REGION Network 10: Example — Equations
   // ▀▀▀▀▀▀▀▀▀▀▀▀▀▀▀▀▀▀▀▀▀▀▀▀▀▀▀▀▀▀▀▀▀▀▀▀▀▀▀▀▀▀▀▀
   // 
   // TITLE:    EQUATIONS (EXAMPLES)
   // 
   // ▄▄▄▄▄▄▄▄▄▄▄▄▄▄▄▄▄▄▄▄▄▄▄▄▄▄▄▄▄▄▄▄▄▄▄▄▄▄▄▄▄▄▄▄
   // 
   // 
   // 
   // ┌─────────────────────────────────────┐
   // │                                                                                                              100                         │
   // │ SigPercent = (Signal ─ PV_RANGE_MIN) ╳ ---------------------------------------------------------------    │
   // │                    (PV_RANGE_MAX ─ PV_RANGE_MIN)    │
   // └─────────────────────────────────────┘
   // 
   // 
   // ┌───────────────────────┐
   // │        2.5               │
   // │ CalcValOOR = ------------ ╳ (RAW_MAX ─ RAW_MIN)   │
   // │       100               │
   // └───────────────────────┘
   // 
   // Mathematical operators:
   //    Large:  ┼ ─ ╳
   //    Small: + − × ÷ ± ≤ ≥
   // 
   //                ━━━   ⬙⬙⬙⬙⬙⬙   ━━━
   // 
   // 
   // ██████████████ █ █ █ █  END   █ █ █ █ ██████████████
END_REGION

REGION Network 11: Example — Figures
   // ▀▀▀▀▀▀▀▀▀▀▀▀▀▀▀▀▀▀▀▀▀▀▀▀▀▀▀▀▀▀▀▀▀▀▀▀▀▀▀▀▀▀▀▀
   // 
   // TITLE:    FIGURES (EXAMPLES)
   // 
   // ▄▄▄▄▄▄▄▄▄▄▄▄▄▄▄▄▄▄▄▄▄▄▄▄▄▄▄▄▄▄▄▄▄▄▄▄▄▄▄▄▄▄▄▄
   // 
   // 
   // 
   // Some example figures, always pad gaps with an EM-SPACE, where text is used add normal 
   // spaces with either a THREE-PER-EM space or a SIX-PER-EM space — one of these will give an
   // exact alignment.
   // 
   // These figures are included to show what is possible.
   // 
   // 
   // Figures have 1 blank line above and 1 below.
   // 
   //   → ┌────────┐
   // ┌───┤   IDLE   │
   // │   └───┬────┘
   // │       ↓
   // │       START
   // │       │
   // │   ┌───┴────┐ →
   // │   │  STARTING     ├───┐
   // │   └───┬────┘   │
   // │       ↓        │
   // │         Run*       ├────────────────────┐
   // │       │        │                    │
   // │   ┌───┴────┐ → │                    │
   // │   │        ├───┴───  Hold  ───┐          │
   // │   │        │             ↓          ↓
   // │   │        │         ┌───┴────┐ ┌───┴────┐
   // │   │        │         │  HOLDING    │ │ ErrHOLDING   │
   // │   │        │         └───┬────┘ └───┬────┘
   // │   │        │             Held*        ErrHeld*
   // │   │        │         ┌───┴────┐ ┌───┴────┐
   // │   │        │         │   HELD    │ │  ErrHELD   │
   // │   │  RUNNING     │         └───┬────┘ └───┬────┘
   // │   │        │              Resume         ErrResume
   // │   │        │         ┌───┴────┐ ┌───┴────┐
   // │  ┌┤        │         │   RESUMING    │ │  ErrRESUMING   │ 
   // │  ││        │         └───┬────┘ └───┬────┘  
   // │  ││        │             │          │
   // │  ││        │ ←           ↓          ↓
   // │  ││        │─────────────┴──────────┘
   // │  │└───┬────┘   Returns to previous step (running or starting)
   // │  ↓    ↓
   // │  │    │
   // │ Complete Complete*     Note: *indicates that the command is issued
   // │  │    │           automatically by the sequence (it
   // │  │┌───┴────┐      can also be triggered manually):
   // │  └┤ COMPLETING  │          1. Run
   // │   └───┬────┘          2. Complete
   // │       ↓               3. Completed
   // ↑     Completed*              4. Held
   // │       │               5. ErrHeld
   // │   ┌───┴────┐          6. Stopped
   // │   │  COMPLETED   │          7. Aborted
   // │   └───┬────┘
   // │       │
   // │              RetIdle*
   // │   ←   ↓
   // ├───────┘
   // │   
   // │
   // │     ABORT ROUTE                  STOPPING ROUTE
   // │Can be triggered in all states except       Can be triggered in all states except
   // │ IDLE, COMPLETED, ABORTING or            IDLE, COMPLETED, ABORTING, 
   // │       ABORTED                 ABORTED, STOPPING or STOPPED
   // │       │                       │
   // │       ↓                       ↓
   // │                Abort                                                                                       Stop
   // │       │                       │
   // │   ┌───┴────┐              ┌───┴────┐
   // ↑   │ ABORTING    │              │  STOPPING    │
   // │   └───┬────┘              └───┬────┘
   // │       ↓                       ↓
   // │              Aborted*                                                                                Stopped*
   // │       │                       │
   // │   ┌───┴────┐              ┌───┴────┐
   // │   │ ABORTED      │              │ STOPPED   │
   // │   └───┬────┘              └───┬────┘
   // │       │                       │
   // │      RetIdle (*)                                                                               RetIdle (*)
   // │  ←    ↓                       ↓
   // └───────┴───────────────────────┘
   // 
   // 
   // 
   // ▌▌▌▌▌▌▌▌▌▌▌▌▌▌▌▌▌▌   INLINE FIGURES ▐▐▐▐▐▐▐▐▐▐▐▐▐▐▐▐▐▐
   // 
   // 
   // 
   // ▂▂▂▂▂▂▂▂▂▂▂▂▂▂▂▂▂▂▂▂▂▂▂▂▂▂▂▂▂▂▂▂▂▂▂▂▂▂▂▂▂▂▂▂
   // 1.1     Step operation and phases
   // 
   // 
   //  ┌─────┐  The sequence progresses from one step to the next if the
   //  │Step n        │  transition logic for the step is TRUE. 
   //  └┬────┘                                                                 
   //   │       In this example, STEP n is active and will remain active
   //         --- T n        until its associated transition (T n) becomes TRUE; at this
   //   │       point the sequence will advance to the next step (STEP n+1)
   //  ┌┴────┐  and execute the actions required of this step. The sequence
   //  │Step n+1    │  will remain in this step until its transition condition is
   //  └┬────┘  true, at which point the sequence will advance again.
   //   │                                                                      
   //         --- T n+1      Each step has a step number, this is an integer value in
   //   │       the range 0 to 29999; step numbers are assigned in specific
   //           Ranges for different operating states of the sequence (IDLE,
   //           STARTING, RUNNING &c.).
   // 
   // Within an individual step, the step has three distinct phases and actions can 
   // be attached to any of these phases (externally to the block). The phases are:
   // 
   // INITIALISING (Phs_INIT)                   ┌──────┐
   // This is activated for a single OB1 scan when the step   │INITIALISING   │
   // is first processed (I.e. on the rising edge of the step     └┬─────┘
   // becoming active).                     │      
   //                           ┌┴─────┐ 
   // PROCESSING (Phs_PROC)               │PROCESSING │
   // This is the main phase of the step, it is activated        └┬─────┘
   // immediately following the INITIALISING phase and remains  │       
   // active until the step TRANSITION condition is TRUE. The     --- T n   
   // PROCESSING phase becomes inactive on the rising edge   │     
   // of the TRANSITION condition.              ┌┴─────┐
   //                           │TERMINATING │    
   // TERMINATING (Phs_TERM)               └──────┘    
   // The TERMINATING phase is activated on the rising edge of the TRANSITION
   // condition (the same condition that terminates the PROCESSING phase). The
   // terminating phase is active for a single OB1 scan.
   // 
   // 
   // [ALTERNATIVE]
   //  ┌──────┐ INITIALISING (Phs_INIT)
   //  │INITIALISING   │ This is activated for a single OB1 scan when the step
   //  └┬─────┘ is first processed (I.e. on the rising edge of the step
   //   │       becoming active).
   //  ┌┴─────┐    
   //  │PROCESSING │ PROCESSING (Phs_PROC)
   //  └┬─────┘ This is the main phase of the step, it is activated 
   //   │       immediately following the INITIALISING phase and remains
   //          --- T n       active until the step TRANSITION condition is TRUE. The
   //   │       PROCESSING phase becomes inactive on the rising edge
   //  ┌┴─────┐ of the TRANSITION condition.
   //  │TERMINATING │    
   //  └──────┘
   // 
   // TERMINATING (Phs_TERM)
   // The TERMINATING phase is activated on the rising edge of the TRANSITION
   // condition (the same condition that terminates the PROCESSING phase). The
   // terminating phase is active for a single OB1 scan.
   // 
   // 
   // 
   // 
   // ▌▌▌▌▌▌▌▌▌▌▌▌▌▌▌▌▌   GRAPHICAL FIGURE   ▐▐▐▐▐▐▐▐▐▐▐▐▐▐▐▐▐
   // 
   //     No. of scans from start of STEP 1
   //     1      2      3     4      5     6       7      8      9
   //   ┼─┼─┼─┼─┼─┼─┼─┼─┼─┼─┼─┼  ─ ─ ┐
   //                                │
   //   ┌─┐                          │
   //   │ │               Phs_INIT
   //  ─┘ └────────────────────                   
   //   ┼─┼─┼─┼─┼─┼─┼─┼─┼─┼─┼─┼                   
   //  
   //     ┌───┐                       S
   //     │   │           Phs_PROC      T
   //  ───┘   └────────────────       E
   //   ┼─┼─┼─┼─┼─┼─┼─┼─┼─┼─┼─┼       P
   //  
   //         ┌─┐                     1
   //         │ │         TRANSITION
   //  ───────┘ └──────────────
   //   ┼─┼─┼─┼─┼─┼─┼─┼─┼─┼─┼─┼
   // 
   //         ┌─┐
   //         │ │         Phs_TERM      │
   //  ───────┘ └──────────────      │
   //   ┼─┼─┼─┼─┼─┼─┼─┼─┼─┼─┼─┼  ─ ─ ┘
   // 
   // 
   //     1      2      3     4      5     6       7      8      9
   //   ┼─┼─┼─┼─┼─┼─┼─┼─┼─┼─┼─┼  ─ ─ ┐
   //                                │
   //           ┌─┐                  │
   //           │ │       Phs_INIT
   //   ────────┘ └────────────                   
   //   ┼─┼─┼─┼─┼─┼─┼─┼─┼─┼─┼─┼                   
   // 
   //             ┌───┐               S
   //             │   │   Phs_PROC      T
   //  ───────────┘   └────────       E
   //   ┼─┼─┼─┼─┼─┼─┼─┼─┼─┼─┼─┼       P
   //                           
   //                 ┌─┐             2
   //                 │ │ TRANSITION
   //  ───────────────┘ └──────      
   //   ┼─┼─┼─┼─┼─┼─┼─┼─┼─┼─┼─┼
   // 
   //                 ┌─┐
   //                 │ │ Phs_TERM      │
   //  ───────────────┘ └──────      │
   //   ┼─┼─┼─┼─┼─┼─┼─┼─┼─┼─┼─┼  ─ ─ ┘
   // 
   // 
   // 
   // ▌▌▌▌▌▌▌▌▌▌▌▌▌▌▌▌▌▌    PAL LOGO    ▐▐▐▐▐▐▐▐▐▐▐▐▐▐▐▐▐▐
   // 
   //          ⠀⠀⠀⠀⠀⠀⠀⠀⠀⠀⠀⠀⠀⠀⠀⠀⠀⠀⠀⠀⠀⠀⠀⠀⠀⠀⠀⠀⠀⣀⣀⣀
   //       ⠀⠀⠀⠀⠀⠀⠀⠀⠀⠀⠀⠀⠀⠀⠀⠀⠀⠀⠀⠀⠀⠀⠀⠀⠀⠀⠀⣤⣶⣿⣿⣿⣿⣿⣿⣤
   //       ⠀⠀⠀⠀⠀⠀⠀⠀⠀⠀⠀⠀⠀⠀⠀⠀⠀⠀⠀⠀⠀⠀⠀⠀⠀⠀⣶⣿⣿⣿⣿⣿⣿⣿⣿⣿⣶
   //       ⠀⠀⠀⠀⠀⠀⠀⠀⠀⠀⠀⠀⠀⠀⠀⠀⠀⠀⠀⠀⠀⠀⠀⠀⠀⠀⣿⣿⣿⣿⣿⣿⣿⣿⣿⣿⣿
   //       ⠀⠀⠀⠀⠀⠀⠀⠀⠀⠀⠀⠀⠀⠀⠀⠀⠀⠀⠀⠀⠀⠀⠀⠀⠀⣀⠛⣿⣿⣿⣿⣿⣿⣿⣿⣿⠿
   //       ⠀⠀⠀⠀⠀⠀⠀⠀⠀⠀⠀⠀⠀⠀⠀⠀⠀⠀⠀⠀⠀⠀⣀⣶⣿⣿⣤⠉⠿⣿⣿⣿⣿⣿⠿⠛⣤⣶
   //       ⠀⠀⠀⠀⠀⠀⠀⠀⠀⠀⠀⠀⠀⠀⠀⠀⠀⠀⠀⠀⣤⣿⣿⣿⣿⣿⣿⣿⣶⣤⠉⠉⠉⠀⠤⣿⣿⣿⣿⣶⣀⣀⣀⣀⣀⣀⣀⣀
   //       ⠀⠀⠀⠀⠀⠀⠀⠀⠀⠀⠀⠀⠀⠀⠀⠀⠀⣀⣶⣿⣿⣿⣿⣿⣿⣿⣿⣿⣿⠉⠀⠀⠀⠀⠀⠉⠿⣿⣿⣿⣿⣿⣿⣿⣿⣿⣿⣿⣶
   //       ⠀⠀⠀⠀⠀⠀⠀⠀⠀⠀⠀⠀⠀⠀⠀⠀⠛⠿⣿⣿⣿⣿⣿⣿⣿⣿⣿⠿⠀⠀⠀⠀⠀⠀⠀⠀⠀⣿⣿⣿⣿⣿⣿⣿⣿⠿⠿⣿⣿⣤
   //       ⠀⠀⠀⠀⠀⠀⠀⠀⠀⣀⣤⣶⣿⣿⣿⣿⣶⣶⣤⠉⠿⣿⣿⣿⣿⣿⠛⠀⠀⠀⠀⠀⠀⠀⠀⠀⠀⣿⣿⣿⣿⠉⠀⠀⠀⠀⠀⠉⣿⣿⣤
   //       ⠀⠀⠀⠀⠀⠀⠀⣀⣶⣿⣿⣿⣿⣿⣿⣿⣿⣿⣿⣿⣤⠉⣿⣿⣿⠛⠀⠀⠀⠀⠀⠀⠀⠀⠀⠀⣿⣿⣿⣿⣿⠀⠀⠀⠀⠀⠀⠀⠀⠿⠿
   //       ⠀⠀⠀⠀⠀⠀⣀⣿⣿⣿⣿⣿⣿⣿⣿⣿⣿⣿⣿⣿⣿⣿⠀⣿⠉⠀⠀⠀⠀⠀⠀⠀⠀⠀⠀⠀⣿⣿⣿⣿⣿
   //       ⠀⠀⠀⠀⠀⠀⣿⣿⣿⣿⣿⣿⣿⣿⣿⣿⣿⣿⣿⣿⣿⣿⣀⠀⠀⠀⠀⠀⠀⠀⠀⠀⠀⠀⠀⠀⠉⠛⠿⣿⣿⣿⣤
   //       ⠀⠀⠀⠀⠀⠀⣿⣿⣿⣿⣿⣿⣿⣿⣿⣿⣿⣿⣿⣿⣿⣿⠿⠀⠀⠀⠀⠀⠀⠀⠀⠀⠀⠀⠀⠀⠀⠀⠀⠀⠉⠛⠿⣿
   //       ⠀⠀⠀⠀⠀⠀⠛⣿⣿⣿⣿⣿⣿⣿⣿⣿⣿⣿⣿⣿⣿⣿
   //       ⠀⠀⠀⠀⠀⠀⠀⠛⣿⣿⣿⣿⣿⣿⣿⣿⣿⣿⣿⣿⠿⠉
   //       ⠀⠀⠀⠀⠀⠀⠀⠀⠀⠛⠿⣿⣿⣿⣿⣿⣿⣿⠿⠉
   //       ⠀⠀⠀⠀⠀⠀⠀⠀⠀⠀⠀⣀⣉⣉⣉⣉⣉⣀
   //       ⠀⠀⠀⠀⠀⠀⠀⠀⠀⣤⣿⣿⣿⣿⣿⣿⣿⣿⣀⠛⣿⣿⣿⣿⣿⣿⣿⣿⣿⣿⣿⣿⣿⣿⣿⣿⣿⣿⣿⣿⣿⣿⣿⣿⣿⣿⣿⣿⣿⣶⣤⣀⠀⠀⠀⠀
   //       ⠀⠀⠀⠀⠀⠀⠀⠀⣤⣿⣿⣿⠿⠉⠉⣿⣿⣿⣿⣤⠉⠿⠿⠿⠿⠿⠿⠿⠿⠿⠿⠿⠿⠿⠿⠿⠿⠿⠿⠿⠿⠿⠿⠿⠿⠿⠿⣿⣿⣿⣿⣿⣿⣀⠀⠀
   //       ⠀⠀⠀⠀⠀⠀⠀⣶⣿⣿⣿⠛⠀⠀   ⠀⠀⠿⣿⣿⣿⣤⠀⠀⠀⠀⠀⠀⣶⣶⣶⣶⣤⠀⠀⠀⠀ ⣶⣶⣶         ⣶⣶⠀⠀⠀⠀⠀⠿⣿⣿⣿⣿⣶⠀
   //       ⠀⠀⠀⠀⠀⠀⣿⣿⣿⣿⠛⠀⠀⠀⠀   ⠀⠀⠛⣿⣿⣿⣶⠀⠀⠀⠀⠀⣿⣿⣿⠿⣿⣿⠀⠀⣤⣿⣿⣿⣤       ⣿⣿⠀⠀⠀⠀⠀⠀ ⠿⣿⣿⣿⣿⣤
   //       ⠀⠀⠀⠀⠀⣿⣿⣿⣿⠉⠀⠀⠀⠀⠀   ⠀⠀⠀⠛⣿⣿⣿⣿⠀⠀⠀⠀⣿⣿⣿⣶⣿⣿⠀⠀⣿⣿⠉⣿⣿       ⣿⣿⠀⠀⠀⠀⠀     ⣿⣿⣿⣿⣿
   //       ⠀⠀⠀⣀⣿⣿⣿⣿⠉⠀⠀⠀⠀⠀⠀⠀⠀   ⠀⠀⠉⣿⣿⣿⣿      ⣿⣿⣿⠛⠛⠀⠀⣶⣿⣿⣿⣿⣿⣶    ⣿⣿⣤⣤⣤      ⣶⣿⣿⣿⣿⠛
   //       ⠀⠀⣤⣿⣿⣿⣿⠉⠀⠀⠀⠀⠀⠀⠀⠀⠀⠀⠀   ⠀⠉⣿⣿⣿⣿⣀ ⠿⠿⠿⠀⠀⠀   ⠿⠿⠉⠉⠉⠿⠿    ⠿⠿⠿⠿⠿ ⠀⣶⣿⣿⣿⣿⠿⠀
   //       ⠀⣤⣿⣿⣿⣿⣿⣶⣤⣤⣤⣤⣤⣤⣤⣤⣤⣤⣤⣤⣶⣿⣿⣿⣿⣿⣀⠀⣶⣶⣶⣶⣶⣶⣶⣶⣶⣶⣶⣶⣶⣶⣶⣶⣶⣶⣶⣶⣿⣿⣿⣿⠉⠀⠀
   //       ⠀⣿⣿⣿⣿⣿⣿⣿⣿⣿⣿⣿⣿⣿⣿⣿⣿⣿⣿⣿⣿⣿⣿⣿⣿⣿⣿⠀⠉⣿⣿⣿⣿⣿⣿⣿⣿⣿⣿⣿⣿⣿⣿⣿⣿⣿⣿⣿⣿⠿⠛⠉⠀⠀⠀⠀
   //       ⠀⠉⠛⠛⠛⠛⠛⠛⠛⠛⠛⠛⠛⠛⠛⠛⠛⠛⠛⠛⠛⠛⠛⠛⠛⠛⠉⠀⠀⠉⠉⠉⠉⠉⠉⠉⠉⠉⠉⠉⠉⠉⠉⠉⠉⠉⠉⠉⠀⠀⠀⠀⠀⠀⠀⠀
   // 
   //                ━━━   ⬙⬙⬙⬙⬙⬙   ━━━
   // 
   // 
   // ██████████████ █ █ █ █  END   █ █ █ █ ██████████████
END_REGION

REGION Network 12: Special characters — Hyphens, whitespace and construction lines
   // ▀▀▀▀▀▀▀▀▀▀▀▀▀▀▀▀▀▀▀▀▀▀▀▀▀▀▀▀▀▀▀▀▀▀▀▀▀▀▀▀▀▀▀▀
   // 
   // TITLE:    SPECIAL CHARACTERS
   // 
   // ▄▄▄▄▄▄▄▄▄▄▄▄▄▄▄▄▄▄▄▄▄▄▄▄▄▄▄▄▄▄▄▄▄▄▄▄▄▄▄▄▄▄▄▄
   // 
   // 
   // The TIA Portal Basic font contains many different types of characters:
   // 
   //    •   Hyphens and whitespace characters
   //    •   Construction lines (these are specially ordered characters, useful for building tables &c.)
   //    •   Arrows
   //    •   Box characters (for drawing box and line diagrams)
   //    •   Block characters
   //    •   Currency
   //    •   Punctuation (extended list)
   //    •   Non-proportional letters and numbers
   //    •   Greek characters
   //    •   Indexing characters
   //    •   Roman numerals
   //    •   Mathematical characters
   //    •   Geometric characters
   //    •   Dingbat characters
   // 
   // The following sections contain a list of these characters for use in TIA Portal comment fields.
   // 
   // Note:    The following tables of characters break the rules for comment fields by exceeding
   //      the prescribed comment field width of 44 em-spaces. This is done to give the 
   //      characters in a more concise form whilst maintaining reasonable descriptions for
   //      the characters
   // 
   // 
   // 
   // ▄▄▄▄▄▄▄▄▄▄▄▄▄▄▄▄▄▄▄▄▄▄▄▄▄▄▄▄▄▄▄▄▄▄▄▄▄▄▄▄▄▄▄▄
   // HYPHENS AND WHITESPACE CHARACTERS
   // 
   // 
   // — Em Dash               █ █ Em Space
   // –   En Dash              █ █   En Space
   // ‐    Hyphen               █ █    Three-Per-Em Space
   // ¬   Soft Hyphen             █ █    Normal Space
   //                       █ █     Six-Per-Em Space
   // 
   // 
   // 
   // ▄▄▄▄▄▄▄▄▄▄▄▄▄▄▄▄▄▄▄▄▄▄▄▄▄▄▄▄▄▄▄▄▄▄▄▄▄▄▄▄▄▄▄▄
   // CONSTRUCTION LINES AND USEFUL LINES
   // 
   // 
   // [Copyable whitespace]
   //  █ █ █ █ █ Em En ThreePerEm SixPerEM
   // [Em-space construction line]
   // ▀▄▀▄▀▄▀▄▀▄▀▄▀▄▀▄▀▄▀▄▀▄▀▄▀▄▀▄▀▄▀▄▀▄▀▄▀▄▀▄▀▄▀▄
   // [Central header — used for examples]
   // ▌▌▌▌▌▌▌▌▌▌▌▌▌▌▌▌▌▌▌▌▌▌▐▐▐▐▐▐▐▐▐▐▐▐▐▐▐▐▐▐▐▐▐▐
   // [Title start]
   // ▀▀▀▀▀▀▀▀▀▀▀▀▀▀▀▀▀▀▀▀▀▀▀▀▀▀▀▀▀▀▀▀▀▀▀▀▀▀▀▀▀▀▀▀
   // [Title end/section over-line]
   // ▄▄▄▄▄▄▄▄▄▄▄▄▄▄▄▄▄▄▄▄▄▄▄▄▄▄▄▄▄▄▄▄▄▄▄▄▄▄▄▄▄▄▄▄
   // [Subsection over-line]
   // ▂▂▂▂▂▂▂▂▂▂▂▂▂▂▂▂▂▂▂▂▂▂▂▂▂▂▂▂▂▂▂▂▂▂▂▂▂▂▂▂▂▂▂▂
   // [Inline section over-line]
   // ▁▁▁▁▁▁▁▁▁▁▁▁▁▁▁▁▁▁▁▁▁▁▁▁▁▁▁▁▁▁▁▁▁▁▁▁▁▁▁▁▁▁▁▁
   // [Table row line]
   //  ――――――――――――――――――――――――――――――――――――――――――
   // [Revision row line]
   //  ―――――――――――――――――――――――――――――――――――――――――――
   // [Flourish divider]
   //                ━━━   ⬙⬙⬙⬙⬙⬙   ━━━
   // [End line]
   // ██████████████ █ █ █ █  END   █ █ █ █ ██████████████
END_REGION

REGION Network 13: Special characters — Arrows, box and block characters
   // ▄▄▄▄▄▄▄▄▄▄▄▄▄▄▄▄▄▄▄▄▄▄▄▄▄▄▄▄▄▄▄▄▄▄▄▄▄▄▄▄▄▄▄▄
   // ARROWS
   // 
   // 
   // ← Left Arrow              ⇐ Left dbl Arrow             ↩ Left Arrow Hook
   // ↑ Up Arrow               ⇑ Up dbl Arrow               ↪ Right Arrow Hook
   // → Right Arrow              ⇒ Right dbl Arrow           ⤣ North West Arrow Hook
   // ↓ Down Arrow             ⇓ Down dbl Arrow             ⤤ North East Arrow Hook
   // ↔ Left Right Arrow             ⇔ Left Right dbl Arrow          ⤥ South East Arrow Hook
   // ↕ Up Down Arrow          ⇕ Up Down dbl Arrow          ⤦ South West Arrow Hook
   // ↖ North West Arrow          ⇖ North West dbl Arrow         ↰    Up Arrow Tip Left
   // ↗ North East Arrow          ⇗ North East dbl Arrow          ↱    Up Arrow Tip Right
   // ↘ South East Arrow          ⇘ South East dbl Arrow         ↲    Down Arrow Tip Left
   // ↙ South West Arrow         ⇙    South West dbl Arrow        ↳ Down Arrow Tip Right
   // ⤡ North West & South East Arrow    ⤂ Left dbl Arrow vert Stroke       ↴ Right Arrow Corner down
   // ⤢ North East & South West Arrow    ⤃ Right dbl Arrow vert Stroke     ↵ Down Arrow Corner Left
   // ⇄ Right Arrow Over Left Arrow       ⤆ Left dbl Arrow From Bar        ↶ Anticlockwise Top Semicircle Arrow
   // ⇅ Up Arrow Left Of down Arrow        ⤇ Right dbl Arrow From Bar         ↷ Clockwise Top Semicircle Arrow
   // ⇆ Left Arrow Over Right Arrow       ⤄ Left Right dbl Arrow vert Stroke    ↺ Anticlockwise Open Circle Arrow
   // ⇇ Left Paired Arrows           ↼ Left Harpoon Barb up         ↻ Clockwise Open Circle Arrow
   // ⇈ Up Paired Arrows             ↽ Left Harpoon Barb down         ⟲ Anticlockwise Gapped Circle Arrow
   // ⇉ Right Paired Arrows         ↾ Up Harpoon Barb Right         ⟳ Clockwise Gapped Circle Arrow
   // ⇊ Down Paired Arrows           ↿ Up Harpoon Barb Left
   // ↤ Left Arrow From Bar           ⇀ Right Harpoon Barb up         ▲  Black Up Triangle 
   // ↥ Up Arrow From Bar          ⇁ Right Harpoon Barb down       ▼  Black Down Triangle
   // ↦ Right Arrow From Bar         ⇂ Down Harpoon Barb Right      ▶  Black Right Triangle
   // ↧ down Arrow From Bar        ⇃ Down Harpoon Barb Left         ◀  Black Left Triangle
   // ↨ Up Down Arrow Base         ⇋ Left Harpoon Over Right Harpoon
   // ↞ Left Two head Arrow          ⇌ Right Harpoon Over Left Harpoon
   // ↟ up Two head Arrow         ↯ Down Zigzag Arrow
   // ↠ Right Two head Arrow
   // ↡ Down Two head Arrow
   // ⤙ Left Arrow-Tail
   // ⤚ Right Arrow-Tail
   // ⤛ Left dbl Arrow-Tail    
   // ⤜ Right dbl Arrow-Tail    
   // ⤝ Left Arrow To Black Diamond    
   // ⤞ Right Arrow To Black Diamond    
   // 
   // ⟵  Long Left Arrow             ↢ Left Arrow Tail             ⌃   Up Arrowhead
   // ⟶  Long Right Arrow          ↣ Right Arrow Tail             ⌄   Down Arrowhead
   // ⟷  Long Left Right Arrow         ⤟ Left Arrow Bar To Black Diamond   ⌅   Projective
   // ⟸  Long Left dbl Arrow         ⤠ Right Arrow Bar To Black Diamond    ⌆   Perspective
   // ⟹  Long Right dbl Arrow          ⤌    Left dbl Dash Arrow         ⟰ Up Quadruple Arrow
   // ⟺  Long Left Right dbl Arrow        ⤍    Right dbl Dash Arrow         ⟱ Down Quadruple Arrow
   // ⟻  Long Left Arrow From Bar       ⤎    Left Triple Dash Arrow        ⤊ Up Triple Arrow
   // ⟼  Long Right Arrow From Bar        ⤏    Right Triple Dash Arrow         ⤋ Down Triple Arrow
   // ⟽  Long Left dbl Arrow From Bar       ⤈    Down Arrow horiz Stroke          ⤈   Down Arrow horiz Stroke
   // ⟾  Long Right dbl Arrow From Bar    ⤉    Up Arrow horiz Stroke             ⤉   Up Arrow horiz Stroke
   // 
   // 
   // 
   // ▄▄▄▄▄▄▄▄▄▄▄▄▄▄▄▄▄▄▄▄▄▄▄▄▄▄▄▄▄▄▄▄▄▄▄▄▄▄▄▄▄▄▄▄
   // BOX CHARACTERS
   // 
   // 
   // ─ Box Light horiz            ╌ Box Light dbl Dash horiz       ⋮     Vert Ellipsis
   // │ Box Light vert             ╎ Box Light dbl Dash vert        ⋯    Midline horiz Ellipsis
   // ╱ Box Light diag top Right Left      ╍ Box Heavy dbl Dash horiz       ⋰     Up Right diag Ellipsis
   // ╲ Box Light diag top Left To btm Right    ╏ Box Heavy dbl Dash vert          ⋱    Down Right diag Ellipsis
   // ╳ Box Light diag Cross          ┄ Box Light Triple Dash horiz      ╴ Box Light Left
   // ━ Box Heavy horiz             ┆ Box Light Triple Dash vert       ╵ Box Light Up
   // ┃ Box Heavy vert           ┅ Box Heavy Triple Dash horiz       ╶ Box Light Right
   // ═ Box dbl horiz               ┇ Box Heavy Triple Dash vert        ╷ Box Light Down
   // ║ Box dbl vert              ┈ Box Light Quadruple Dash horiz     ╸ Box Heavy Left
   //                       ┊ Box Light Quadruple Dash vert       ╹ Box Heavy Up
   //                       ┉ Box Heavy Quadruple Dash horiz      ╺ Box Heavy Right
   //                       ┋ Box Heavy Quadruple Dash vert     ╻ Box Heavy Down
   // 
   // ┌ Box Light Down & Right        ├ Box Light vert & Right         ─ Box Light horiz
   // └ Box Light Up & Right           ┤ Box Light vert & Left        │ Box Light vert
   // ┐ Box Light Down & Left           ┬ Box Light Down & horiz         ┼ Box Light vert & horiz
   // ┘ Box Light Up & Left          ┴ Box Light Up & horiz  
   // ┏ Box Heavy Down & Right         ┣ Box Heavy vert & Right          ━ Box Heavy horiz
   // ┗ Box Heavy Up & Right         ┫ Box Heavy vert & Left         ┃ Box Heavy vert
   // ┓ Box Heavy Down & Left         ┳ Box Heavy Down & horiz       ╋ Box Heavy vert & horiz
   // ┛ Box Heavy Up & Left        ┻ Box Heavy Up & horiz  
   //     
   // ┍ Box Down Light & Right Heavy     ┝ Box vert Light & Right Heavy      ━ Box Heavy horiz
   // ┕ Box Up Light & Right Heavy        ┥ Box vert Light & Left Heavy     │ Box Light vert
   // ┑ Box Down Light & Left Heavy     ┯ Box Down Light & horiz Heavy      ┿ Box vert Light & horiz Heavy
   // ┙ Box Up Light & Left Heavy       ┷ Box Up Light & horiz Heavy  
   // 
   // ┎ Box Down Heavy & Right Light     ┠ Box vert Heavy & Right Light      ─ Box Light horiz
   // ┖ Box Up Heavy & Right Light        ┨ Box vert Heavy & Left Light     ┃ Box Heavy vert
   // ┒ Box Down Heavy & Left Light     ┰ Box Down Heavy & horiz Light      ╂ Box vert Heavy & horiz Light
   // ┚ Box Up Heavy & Left Light       ┸ Box Up Heavy & horiz Light  
   // 
   // ┦ Box Up Heavy & Left Down Light     ┪ Box Up Light & Left Down Heavy     ╀ Box Up Heavy & Down horiz Light
   // ┶ Box Right Heavy & Left Up Light   ┹ Box Right Light & Left Up Heavy   ┾ Box Right Heavy & Left vert Light
   // ┟ Box Down Heavy & Right Up Light     ┡ Box Down Light & Right Up Heavy     ╁ Box Down Heavy & Up horiz Light
   // ┭ Box Left Heavy & Right Down Light    ┲ Box Left Light & Right Down Heavy    ┽ Box Left Heavy & Right vert Light
   //  
   // ┞ Box Up Heavy & Right Down Light     ┢ Box Up Light & Right Down Heavy     ╈ Box Up Light & Down horiz Heavy
   // ┮ Box Right Heavy & Left Down Light    ┱ Box Right Light & Left Down Heavy    ╉ Box Right Light & Left vert Heavy
   // ┧ Box Down Heavy & Left Up Light     ┩ Box Down Light & Left Up Heavy     ╇ Box Down Light & Up horiz Heavy
   // ┵ Box Left Heavy & Right Up Light      ┺ Box Left Light & Right Up Heavy   ╊ Box Left Light & Right vert Heavy
   // 
   // ╼ Box Light Left & Heavy Right                            ╄ Box Right Up Heavy & Left Down Light
   // ╽ Box Light Up & Heavy Down                            ╆ Box Right Down Heavy & Left Up Light
   // ╾ Box Heavy Left & Light Right                            ╅ Box Left Down Heavy & Right Up Light
   // ╿ Box Heavy Up & Light Down                            ╃ Box Left Up Heavy & Right Down Light
   // 
   // ╔ Box dbl Down & Right         ╠ Box dbl vert & Right         ═ Box dbl horiz
   // ╚ Box dbl Up & Right           ╣ Box dbl vert & Left           ║ Box dbl vert
   // ╗ Box dbl Down & Left        ╦ Box dbl Down & horiz         ╬ Box dbl vert & horiz
   // ╝ Box dbl Up & Left          ╩ Box dbl Up & horiz  
   //  
   // ╒ Box Down Single & Right dbl     ╞ Box vert Single & Right dbl      ═ Box dbl horiz
   // ╘ Box Up Single & Right dbl        ╡ Box vert Single & Left dbl        │ Box Light vert
   // ╕ Box Down Single & Left dbl        ╤ Box Down Single & horiz dbl      ╪ Box vert Single & horiz dbl
   // ╛ Box Up Single & Left dbl       ╧ Box Up Single & horiz dbl  
   // 
   // ╓ Box Down dbl & Right Single     ╟ Box vert dbl & Right Single      ─ Box Light horiz
   // ╙ Box Up dbl & Right Single        ╢ Box vert dbl & Left Single        ║ Box dbl vert
   // ╖ Box Down dbl & Left Single        ╥ Box Down dbl & horiz Single      ╫ Box vert dbl & horiz Single
   // ╜ Box Up dbl & Left Single       ╨ Box Up dbl & horiz Single  
   // 
   // 
   // 
   // ▄▄▄▄▄▄▄▄▄▄▄▄▄▄▄▄▄▄▄▄▄▄▄▄▄▄▄▄▄▄▄▄▄▄▄▄▄▄▄▄▄▄▄▄
   // BLOCK CHARACTERS
   // 
   // 
   // ▀ Top Half Block             ❘    Light vert Bar              ❘ ❘     En Space
   // ▄ Btm Half Block            ❙    Medium vert Bar           ❘ ❘   Em Space
   // ▐ Right Half Block          ❚   Heavy vert Bar  
   // ▌ Left Half Block    
   // 
   // ▔ Top One Eighth Block        ▉ Left Seven Eighths Block
   // ▁ Btm One Eighth Block          ▊ Left Three Quarters Block
   // ▂ Btm One Quarter Block        ▋ Left Five Eighths Block
   // ▃ Btm Three Eighths Block      ▌ Left Half Block
   // ▄ Btm Half Block            ▍ Left Three Eighths Block
   // ▅ Btm Five Eighths Block         ▎ Left One Quarter Block
   // ▆ Btm Three Quarters Block       ▏ Left One Eighth Block
   // ▇ Btm Seven Eighths Block        ▕ Right One Eighth Block
   // █ Full Block
   // ░ Light Shade
   // ▒ Medium Shade    
   // ▓ Dark Shade    
   // 
   // 
   // ██████████████ █ █ █ █  END   █ █ █ █ ██████████████
END_REGION

REGION Network 14: Special characters — Currency, punctuation and full-width characters
   // ▄▄▄▄▄▄▄▄▄▄▄▄▄▄▄▄▄▄▄▄▄▄▄▄▄▄▄▄▄▄▄▄▄▄▄▄▄▄▄▄▄▄▄▄
   // CURRENCY
   // 
   // 
   // ₳   Austral Sign             €   Euro Sign              ₦  Naira Sign
   // ₵   Cedi Sign               ₠  Euro-Currency Sign          ₪  New Shekel Sign
   // ¢   Cent Sign              ₣  French Franc Sign           ₧   Peseta Sign
   // ₡   Colon Sign               ₰   German Penny Sign           ₱   Peso Sign
   // ₢   Cruzeiro Sign           ₲   Guarani Sign              £  Pound Sign
   // ¤  Currency Sign             ₴   Hryvnia Sign            ₨    Rupee Sign
   // $   Dollar Sign            ₭   Kip Sign              ₮   Tugrik Sign
   // ₫   Dong Sign             ₤   Lira Sign             ₩  Won Sign
   // ₯ Drachma Sign            ₥  Mill Sign              ¥   Yen Sign
   // 
   // 
   // 
   // ▄▄▄▄▄▄▄▄▄▄▄▄▄▄▄▄▄▄▄▄▄▄▄▄▄▄▄▄▄▄▄▄▄▄▄▄▄▄▄▄▄▄▄▄
   // PUNCTUATION AND COMMON SYMBOLS
   // 
   // 
   // #  Hash Sign             "   Quote                 §   Section Sign
   // $   Dollar Sign            “    Left dbl quote             ¶   Pilcrow Sign
   // %  Percent Sign            ”    Right dbl quote
   // &   Ampersand             '    Apostrophe  
   // *   Asterisk              ‘    Left Single quote          †   Dagger
   // ~   Tilde                 ’    Right Single quote           ‡   Dbl Dagger
   // +   Plus Sign               ‹    Single Left Angle quote       •   Bullet
   // -    Hyphen/minus            ›    Single Right Angle quote        ·    Middle Dot
   // =   Equals Sign                                ‣   Triangular Bullet
   // <   Less-Than Sign           ´   Acute Accent              ⁃    Hyphen Bullet
   // >   Greater-Than Sign           `   Grave Accent
   // (    Left Parenthesis
   // )    Right Parenthesis            ©  Copyright Sign           ⁎   Low Asterisk
   // [    Left Square Bracket           ®  Registered Sign  
   // ]    Right Square Bracket         ℀  Account Of               ․    One Dot Leader
   // {   Left Curly Bracket          ℁  Addressed To The Subject      ‥   Two Dot Leader
   // }   Right Curly Bracket          ℂ  Dbl-Struck Capital C           …  Horiz Ellipsis
   // 〈    Left Angle Bracket           ℄   Centre Line Symbol  
   // 〉    Right Angle Bracket            ℅  Care Of               ※  Reference Mark
   // ⁅    Left Square Bracket Quill        ℗  Sound Recording Copyright       ‼   Dbl Exclamation Mark
   // ⁆    Right Square Bracket Quill      ™  Trade Mark Sign            ‽   Interrobang
   // ,    Comma                                 ⁇  Dbl Question Mark
   // .    Full Stop                                   ⁈   Question Exclamation Mark
   // :    Colon                                  ⁉  Exclamation Question Mark
   // ;    Semicolon    
   // !    Exclamation Mark            ⁑   Two Asterisks Aligned vertically     |    Vert Line
   // ?   Question Mark           ⁂   Asterism               ¦    Broken Bar
   // @  Commercial At                              ‖    Dbl vert Line
   // ^   Circumflex Accent            ⁀  Character Tie              ‗   Dbl Low Line
   // /    Solidus               ‿  Undertie             ⁞    Vert Four Dots
   // \    Reverse Solidus            ⁐  Close Up
   // _   Underscore
   // ― Horiz Bar    
   // ¯   Macron
   // ‾   Overline
   // 
   // 
   // 
   // ▄▄▄▄▄▄▄▄▄▄▄▄▄▄▄▄▄▄▄▄▄▄▄▄▄▄▄▄▄▄▄▄▄▄▄▄▄▄▄▄▄▄▄▄
   // NON-PROPORTIONAL (FULL-WIDTH) LETTERS
   // 
   // 
   // Ａ Fullwidth Capital Letter A        ａ Fullwidth Small Letter A       ＂ Fullwidth quote
   // Ｂ Fullwidth Capital Letter B        ｂ Fullwidth Small Letter B       ＇ Fullwidth Apostrophe
   // Ｃ Fullwidth Capital Letter C        ｃ Fullwidth Small Letter C       ＃ Fullwidth Number Sign
   // Ｄ Fullwidth Capital Letter D       ｄ Fullwidth Small Letter D       ＄ Fullwidth Dollar Sign
   // Ｅ Fullwidth Capital Letter E        ｅ Fullwidth Small Letter E       ％ Fullwidth Percent Sign
   // Ｆ Fullwidth Capital Letter F        ｆ Fullwidth Small Letter F       ＆ Fullwidth Ampers&
   // Ｇ Fullwidth Capital Letter G       ｇ Fullwidth Small Letter G       ＊ Fullwidth Asterisk
   // Ｈ Fullwidth Capital Letter H       ｈ Fullwidth Small Letter H          ～ Fullwidth Tilde
   // Ｉ Fullwidth Capital Letter I         ｉ Fullwidth Small Letter I        ＋ Fullwidth Plus Sign
   // Ｊ Fullwidth Capital Letter J         ｊ Fullwidth Small Letter J        － Fullwidth Hyphen-Minus
   // Ｋ Fullwidth Capital Letter K        ｋ Fullwidth Small Letter K       ＝ Fullwidth Equals Sign
   // Ｌ Fullwidth Capital Letter L        ｌ Fullwidth Small Letter L       ＜ Fullwidth Less-Than Sign
   // Ｍ Fullwidth Capital Letter M       ｍ Fullwidth Small Letter M         ＞ Fullwidth Greater-Than Sign
   // Ｎ Fullwidth Capital Letter N       ｎ Fullwidth Small Letter N          （ Fullwidth Left Parenthesis
   // Ｏ Fullwidth Capital Letter O       ｏ Fullwidth Small Letter O       ） Fullwidth Right Parenthesis
   // Ｐ Fullwidth Capital Letter P        ｐ Fullwidth Small Letter P       ［ Fullwidth Left Square Bracket
   // Ｑ Fullwidth Capital Letter Q       ｑ Fullwidth Small Letter Q         ］ Fullwidth Right Square Bracket
   // Ｒ Fullwidth Capital Letter R        ｒ Fullwidth Small Letter R       ｛ Fullwidth Left Curly Bracket
   // Ｓ Fullwidth Capital Letter S        ｓ Fullwidth Small Letter S       ｝ Fullwidth Right Curly Bracket
   // Ｔ Fullwidth Capital Letter T        ｔ Fullwidth Small Letter T        ， Fullwidth Comma
   // Ｕ Fullwidth Capital Letter U       ｕ Fullwidth Small Letter U       ． Fullwidth Full Stop
   // Ｖ Fullwidth Capital Letter V        ｖ Fullwidth Small Letter V       ： Fullwidth Colon
   // Ｗ Fullwidth Capital Letter W       ｗ Fullwidth Small Letter W         ； Fullwidth Semicolon
   // Ｘ Fullwidth Capital Letter X        ｘ Fullwidth Small Letter X       ！ Fullwidth Exclamation Mark
   // Ｙ Fullwidth Capital Letter Y        ｙ Fullwidth Small Letter Y       ？ Fullwidth Question Mark
   // Ｚ Fullwidth Capital Letter Z        ｚ Fullwidth Small Letter Z       ＠ Fullwidth Commercial At
   //                                         ＾ Fullwidth Circumflex Accent
   // ０ Fullwidth Digit Zero         ５ Fullwidth Digit Five          ／ Fullwidth Solidus
   // １ Fullwidth Digit One         ６ Fullwidth Digit Six         ＼ Fullwidth Reverse Solidus
   // ２ Fullwidth Digit Two          ７ Fullwidth Digit Seven         ＿ Fullwidth Low Line
   // ３ Fullwidth Digit Three          ８ Fullwidth Digit Eight           ｜ Fullwidth vert Line
   // ４ Fullwidth Digit Four         ９ Fullwidth Digit Nine         ❘ ❘   Fullwidth space    
   // 
   // 
   // ██████████████ █ █ █ █  END   █ █ █ █ ██████████████
END_REGION

REGION Network 15: Special characters — Greek, indexing characters and Roman numerals
   // ▄▄▄▄▄▄▄▄▄▄▄▄▄▄▄▄▄▄▄▄▄▄▄▄▄▄▄▄▄▄▄▄▄▄▄▄▄▄▄▄▄▄▄▄
   // GREEK CHARACTERS
   // 
   // 
   // Α  Greek Capital Letter Alpha        α   Greek Small Letter Alpha
   // Β   Greek Capital Letter Beta       β   Greek Small Letter Beta
   // Γ   Greek Capital Letter Gamma       γ   Greek Small Letter Gamma
   // Δ  Greek Capital Letter Delta      δ   Greek Small Letter Delta
   // Ε   Greek Capital Letter Epsilon     ε   Greek Small Letter Epsilon
   // Ζ   Greek Capital Letter Zeta       ζ   Greek Small Letter Zeta
   // Η  Greek Capital Letter Eta       η   Greek Small Letter Eta
   // Θ  Greek Capital Letter Theta      θ   Greek Small Letter Theta
   // Ι    Greek Capital Letter Iota         ι    Greek Small Letter Iota
   // Κ   Greek Capital Letter Kappa       κ   Greek Small Letter Kappa
   // Λ   Greek Capital Letter Lambda       λ   Greek Small Letter Lambda
   // Μ  Greek Capital Letter Mu       μ   Greek Small Letter Mu
   // Ν  Greek Capital Letter Nu        ν   Greek Small Letter Nu
   // Ξ   Greek Capital Letter Xi         ξ   Greek Small Letter Xi
   // Ο  Greek Capital Letter Omicron      ο   Greek Small Letter Omicron
   // Π  Greek Capital Letter Pi          π   Greek Small Letter Pi
   // Ρ   Greek Capital Letter Rho      ρ   Greek Small Letter Rho
   // Σ   Greek Capital Letter Sigma       ς   Greek Small Letter Final Sigma
   //                       σ   Greek Small Letter Sigma
   // Τ   Greek Capital Letter Tau         τ   Greek Small Letter Tau
   // Υ   Greek Capital Letter Upsilon     υ   Greek Small Letter Upsilon
   // Φ  Greek Capital Letter Phi       φ  Greek Small Letter Phi
   // Χ   Greek Capital Letter Chi       χ   Greek Small Letter Chi
   // Ψ  Greek Capital Letter Psi        ψ  Greek Small Letter Psi
   // 
   // 
   // 
   // ▄▄▄▄▄▄▄▄▄▄▄▄▄▄▄▄▄▄▄▄▄▄▄▄▄▄▄▄▄▄▄▄▄▄▄▄▄▄▄▄▄▄▄▄
   // INDEXING CHARACTERS  (all characters are 1 EM wide)
   // 
   // 
   // ① Circled One              ⑴ Bracketed One           ⒈ One Full Stop
   // ② Circled Two              ⑵ Bracketed Two           ⒉ Two Full Stop
   // ③ Circled Three              ⑶ Bracketed Three           ⒊ Three Full Stop
   // ④ Circled Four             ⑷ Bracketed Four             ⒋ Four Full Stop
   // ⑤ Circled Five              ⑸ Bracketed Five           ⒌ Five Full Stop
   // ⑥ Circled Six             ⑹ Bracketed Six             ⒍ Six Full Stop
   // ⑦ Circled Seven             ⑺ Bracketed Seven          ⒎ Seven Full Stop
   // ⑧ Circled Eight            ⑻ Bracketed Eight            ⒏ Eight Full Stop
   // ⑨ Circled Nine             ⑼ Bracketed Nine          ⒐ Nine Full Stop
   // ⑩ Circled Ten            ⑽ Bracketed Ten            ⒑ Ten Full Stop
   // ⑪ Circled Eleven            ⑾ Bracketed Eleven         ⒒ Eleven Full Stop
   // ⑫ Circled Twelve            ⑿ Bracketed Twelve         ⒓ Twelve Full Stop
   // ⑬ Circled Thirteen             ⒀ Bracketed Thirteen          ⒔ Thirteen Full Stop
   // ⑭ Circled Fourteen           ⒁ Bracketed Fourteen        ⒕ Fourteen Full Stop
   // ⑮ Circled Fifteen            ⒂ Bracketed Fifteen         ⒖ Fifteen Full Stop
   // ⑯ Circled Sixteen           ⒃ Bracketed Sixteen           ⒗ Sixteen Full Stop
   // ⑰ Circled Seventeen           ⒄ Bracketed Seventeen        ⒘ Seventeen Full Stop
   // ⑱ Circled Eighteen           ⒅ Bracketed Eighteen        ⒙ Eighteen Full Stop
   // ⑲ Circled Nineteen           ⒆ Bracketed Nineteen           ⒚ Nineteen Full Stop
   // ⑳ Circled Twenty            ⒇ Bracketed Twenty         ⒛ Twenty Full Stop
   // 
   // 
   // 
   // ▄▄▄▄▄▄▄▄▄▄▄▄▄▄▄▄▄▄▄▄▄▄▄▄▄▄▄▄▄▄▄▄▄▄▄▄▄▄▄▄▄▄▄▄
   // ROMAN NUMERALS
   // 
   // 
   // Ⅰ    Roman num One          ⅰ    Small Roman num One
   // Ⅱ   Roman num Two           ⅱ   Small Roman num Two
   // Ⅲ  Roman num Three           ⅲ  Small Roman num Three
   // Ⅳ  Roman num Four          ⅳ  Small Roman num Four
   // Ⅴ   Roman num Five          ⅴ   Small Roman num Five
   // Ⅵ  Roman num Six             ⅵ  Small Roman num Six
   // Ⅶ Roman num Seven         ⅶ    Small Roman num Seven
   // Ⅷ    Roman num Eight           ⅷ   Small Roman num Eight
   // Ⅸ  Roman num Nine            ⅸ  Small Roman num Nine
   // Ⅹ   Roman num Ten           ⅹ   Small Roman num Ten
   // Ⅺ  Roman num Eleven           ⅺ  Small Roman num Eleven
   // Ⅻ Roman num Twelve           ⅻ  Small Roman num Twelve
   // Ⅼ   Roman num Fifty           ⅼ    Small Roman num Fifty
   // Ⅽ   Roman num One Hundred        ⅽ   Small Roman num One Hundred
   // Ⅾ  Roman num Five Hundred      ⅾ   Small Roman num Five Hundred
   // Ⅿ  Roman num One Thousand      ⅿ     Small Roman num One Thousand    
   // 
   // 
   // ████████████████████ END    ████████████████████
END_REGION

REGION Network 16: Special characters — Mathematical operators (including vulgar fractions)
   // ▄▄▄▄▄▄▄▄▄▄▄▄▄▄▄▄▄▄▄▄▄▄▄▄▄▄▄▄▄▄▄▄▄▄▄▄▄▄▄▄▄▄▄▄
   // MATHEMATICAL OPERATORS
   // 
   // 
   // ×   Multiplication Sign          ¹   Superscript One           ∅  Empty Set
   // ÷   Division Sign              ²   Superscript Two            ∈  Element Of
   // +   Plus sign                ³   Superscript Three         ∉  Not An Element Of
   // −   Minus Sign            ½  Vulgar Fraction One Half         ∊   Small Element Of
   // ⁒   Commercial Minus Sign       ⅓  Vulgar Fraction One Third       ∋  Contains As Member
   // ±   Plus-Minus Sign             ⅔  Vulgar Fraction Two Thirds      ∌  Does Not Contain As Member
   // ∓   Minus-Or-Plus Sign          ¼  Vulgar Fraction One Quarter        ∍   Small Contains As Member
   // ≤   Less-Than Or Equal To       ¾  Vulgar Fraction Three Quarters      ∩   Intersection
   // ≥   Greater-Than Or Equal To        ⅕  Vulgar Fraction One Fifth        ∪   Union
   // ≪  Much Less-Than            ⅖  Vulgar Fraction Two Fifths       ⊂  Subset Of
   // ≫  Much Greater-Than          ⅗  Vulgar Fraction Three Fifths       ⊃  Superset Of
   // √  Square Root             ⅘  Vulgar Fraction Four Fifths      ⊄  Not A Subset Of
   // ∛  Cube Root             ⅙  Vulgar Fraction One Sixth       ⊅  Not A Superset Of
   // ∜  Fourth Root              ⅚  Vulgar Fraction Five Sixths        ⊆  Subset Of Or Equal To
   // ∝  Proportional To           ⅛  Vulgar Fraction One Eighth       ⊇  Superset Of Or Equal To
   // ∞  Infinity              ⅜  Vulgar Fraction Three Eighths      ⊈  not A Subset Of Nor Equal To
   // °   Degree Sign            ⅝  Vulgar Fraction Five Eighths     ⊉  not A Superset Of Nor Equal To
   // µ   Micro Sign             ⅞  Vulgar Fraction Seven Eighths    ⊊  Subset Of Not Equal To
   // ‰   Per Mille Sign              ⅟   Fraction Numerator One         ⊋  Superset Of Not Equal To
   // ‱  Per Ten Thousand& Sign          ⁄    Fraction Slash            ⊌   Multiset
   // ∀  For All                                    ⊍   Multiset Multiplication
   // ∁   Complement                                 ⊎   Multiset Union
   // ∂   Partial Differential                              ⊏  Square Image Of
   // ∃   There Exists                                ⊐  Square Original Of
   // ∄   There Does Not Exist          ∆   Increment             ⊑  Square Image Of Or Equal To
   // ∴    Therefore               ∇  Nabla               ⊒  Square Original Of Or Equal To
   // ∵    Because                                   ⊓  Square Cap
   // ∶   Ratio                                   ⊔  Square Cup
   // ∷  Proportion    
   // ∿  Sine Wave    
   //      
   // ∥   Parallel To             ∫    Integral               ⌠    Top Half Integral
   // ∦   Not Parallel To            ∬    Dbl Integral              ⌡    Bottom Half Integral
   // ∟ Right Angle              ∭   Triple Integral             ❲   Light Left Shell Bracket 
   // ⊾  Right Angle Arc           ∮   Contour Integral           ❳   Light Right Shell Bracket 
   // ⊿  Right Triangle             ∯    Surface Integral            ⟪   Maths Left dbl Angle Bracket
   // ∠  Angle               ∰   Volume Integral            ⟫   Maths Right dbl Angle Bracket
   // ∡  Measured Angle           ∱   Clockwise Integral           ⟬   Maths Left White Shell Bracket
   // ∢  Spherical Angle            ∲   Clockwise Contour Integral       ⟭   Maths Right White Shell Bracket
   // ⌒    Arc                 ∳   Anticlockwise Contour Integral
   // ⌓    Segment    
   // ⌔     Sector    
   // 
   // ≃   Asymptotically Equal To       ⊕    Circled Plus              ′    Prime
   // ≄   Not Asymptotically Equal To      ⊖    Circled Minus              ″    Dbl Prime
   // ≅   Approx Equal To            ⊗    Circled Times              ‴   Triple Prime
   // ≆   Approx But Not Actually Equal To    ⊘    Circled Division Slash        ⁗   Quadruple Prime
   // ≇   Not approx Nor Actually Equal To   ⊙    Circled Dot Operator          ‵    Reversed Prime
   // ≈   Almost Equal To            ⊚    Circled Ring Operator        ‶    Reversed dbl Prime
   // ≉  Not Almost Equal To          ⊛    Circled Asterisk Operator        ‷   Reversed Triple Prime
   // ≊   Almost Equal Or Equal To       ⊜    Circled Equals
   // ≋   Triple Tilde             ⊝    Circled Dash
   // ≌   All Equal To              ⊞    Squared Plus
   // ≍  Equivalent To             ⊟    Squared Minus
   // ≡   Identical To              ⊠    Squared Times
   // ≢   Not Identical To             ⊡    Squared Dot Operator
   //      
   // ∧  Logical &               ⊢  Right Tack              °   Degree Sign
   // ∨  Logical Or             ⊣  Left Tack                ℃    Degree Celsius
   // ⊻  Xor                 ⊤  Down Tack               ℉    Degree Fahrenheit
   // ⊼  Nand                ⊥  Up Tack                Ω    Ohm Sign    
   // 
   // 
   // ██████████████ █ █ █ █  END   █ █ █ █ ██████████████
END_REGION

REGION Network 17: Special characters — Geometrical and ornamental characters
   // ▄▄▄▄▄▄▄▄▄▄▄▄▄▄▄▄▄▄▄▄▄▄▄▄▄▄▄▄▄▄▄▄▄▄▄▄▄▄▄▄▄▄▄▄
   // GEOMETRICAL CHARACTERS
   // 
   // 
   // ⌉    Right Ceiling            ▬  Black Rectangle            ▭  White Rectangle
   // ⌋    Right Floor                ▮   Black vert Rectangle          ▯   White vert Rectangle
   // ⌈    Left Ceiling               ▰  Black Parallelogram           ▱  White Parallelogram
   // ⌊    Left Floor               ◆  Black Diamond             ◇ White Diamond
   // ⌝   Top Right Corner 
   // ⌟   Bottom Right Corner          ◈  Diamond with Diamond          ◊  Lozenge
   // ⌜   Top Left Corner           ▲  Black Up Triangle             △  White Up Triangle
   // ⌞   Bottom Left Corner          ▶  Black Right Triangle         ▷  White Right Triangle
   // ◝ Top Right quad Circular Arc        ▼  Black Down Triangle          ▽ White Down Triangle
   // ◞ Btm Right quad Circular Arc       ◀  Black Left Triangle           ◁  White Left Triangle
   // ◜ Top Left quad Circular Arc       ▴   Black Up Small Triangle       ▵   White Up Small Triangle
   // ◟ Btm Left quad Circular Arc      ▸   Black Right Small Triangle      ▹   White Right Small Triangle
   // ◘ Inv Bullet               ▾   Black Down Small Triangle     ▿   White Down Small Triangle
   // ◙ Inv White Circle             ◂   Black Left Small Triangle         ◃   White Left Small Triangle
   // ◚ Top Half inv White Circle       ►  Black Right Pointer          ▻  White Right Pointer
   // ◛ Btm Half inv White Circle      ◄  Black Left Pointer          ◅  White Left Pointer
   //      
   // ◻  White Medium Square       ◼  Black Medium Square          ⬔    Square top Right diag Half Black
   // □  White Square              ■  Black Square           ⬕    Square btm Left diag Half Black
   // ◽   White Medium Small Square     ◾   Black Medium Small Square     ⬖    Diamond Left Half Black
   // ▫  White Small Square           ▪  Black Small Square         ⬗    Diamond Right Half Black
   // ▣  Square with Square                              ⬘    Diamond Top Half Black
   // ◉  Fisheye                                  ⬙    Diamond Bottom Half Black
   // ○  White Circle              ●  Black Circle              ◪  Square btm Right diag Half Black
   // ◌  Dotted Circle              ◍  Circle vert Fill              ◫  White Square vert Bisecting Line
   // ◯ Large Circle             ◎ Bullseye              ◬  White Up Triangle Dot
   // ▢  White Square Rounded Corners                        ◭  Up Triangle Left Black
   // ▤  Square horiz Fill                               ◮  Up Triangle Right Black
   // ▥  Square vert Fill                                ◐  Circle Left Half Black
   // ▦  Square Orthogonal Crosshatch Fill   ◖   Left Half Black Circle          ◑  Circle Right Half Black
   // ▧  Square top Left To btm Right Fill     ◗   Right Half Black Circle        ◒  Circle btm Half Black
   // ▨  Square top Right To btm Left Fill                       ◓  Circle top Half Black
   // ▩  Square diag Crosshatch Fill    
   //      
   // ◸    Top Left Triangle                                     ◰    White Square top Left quad
   // ◹    Top Right Triangle                               ◱    White Square btm Left quad
   // ◿    Btm Right Triangle                              ◲    White Square btm Right quad
   // ◺    Btm Left Triangle                                ◳    White Square top Right quad
   // ⧖  White Hourglass           ⧗  Black Hourglass            ◴    White Circle top Left quad
   // ⋈  Bowtie                                         ◵    White Circle btm Left quad
   // 
   // 
   // 
   // ▄▄▄▄▄▄▄▄▄▄▄▄▄▄▄▄▄▄▄▄▄▄▄▄▄▄▄▄▄▄▄▄▄▄▄▄▄▄▄▄▄▄▄▄
   // ORNAMENTAL CHARACTERS
   // 
   // 
   // ⌂  House              ☣  Biohazard Sign           ♚  Black Chess King
   // ⌕  Telephone Recorder           ☤  Caduceus              ♛  Black Chess Queen
   // ⌖   Position Indicator            ☥  Ankh                 ♜  Black Chess Rook
   // ⌗    Viewdata Square          ☮    Peace Symbol            ♝  Black Chess Bishop
   // ⌘    Place Of Interest Sign        ☯ Yin Yang                ♞  Black Chess Knight
   // ⌚     Watch               ☰    Trigram For Heaven           ♟  Black Chess Pawn
   // ⌛  Hourglass             ☱    Trigram For Lake           ♠  Black Spade Suit
   // ⌢  Frown                  ☲    Trigram For Fire             ♡  White Heart Suit
   // ⌣  Smile               ☳    Trigram For Thunder           ♢  White Diamond Suit
   // ⌥  Option Key            ☴    Trigram For Wind           ♣    Black Club Suit
   // ⌦   Erase To The Right           ☵    Trigram For Water            ♤  White Spade Suit
   // ⌧    X In A Rectangle Box          ☶    Trigram For Mountain           ♥  Black Heart Suit
   // ⌨  Keyboard               ☷    Trigram For Earth          ♦  Black Diamond Suit
   // ⌫   Erase To The Left          ☸ Wheel Of Dharma            ♧    White Club Suit
   //                       ☹  White Frowning Face         ♨    Hot Springs
   //                       ☺  White Smiling Face         ♩  Quarter Note
   //                       ☻  Black Smiling Face          ♪  Eighth Note
   // ☀  Black Sun Rays              ☼    White Sun Rays           ♫  Beamed Eighth Notes
   // ☁     Cloud               ☽  First Quarter Moon          ♬  Beamed Sixteenth Notes
   // ☂     Umbrella               ☾  Last Quarter Moon          ♭ Music Flat Sign
   // ☃  Snowman             ☿  Mercury               ♮  Music Natural Sign
   // ☄  Comet                 ♀  Female Sign               ♯ Music Sharp Sign
   // ★  Black Star              ♁  Earth                ⚀ Die Face-1
   // ☆ White Star             ♂    Male Sign              ⚁ Die Face-2
   // ☇   Lightning               ♃  Jupiter                 ⚂ Die Face-3
   // ☈  Thunderstorm            ♄  Saturn                 ⚃ Die Face-4
   // ☉    Sun                ♅  Uranus                ⚄ Die Face-5
   // ☊ Ascending Node           ♆   Neptune             ⚅ Die Face-6
   // ☋ Descending Node           ♇  Pluto                 ⚆ White Circle Dot Right
   // ☌  Conjunction             ♈   Aries                 ⚇ White Circle Two Dots
   // ☍    Opposition               ♉   Taurus                 ⚈ Black Circle White Dot Right
   // ☎   Black Telephone           ♊ Gemini               ⚉ Black Circle Two White Dots
   // ☏   White Telephone           ♋   Cancer                ⚠  Warning Sign
   // ☐  Ballot Box              ♌ Leo                ✁   Top Blade Scissors
   // ☑  Ballot Box Check           ♍ Virgo                ✂   Black Scissors
   // ☒  Ballot Box X              ♎    Libra                 ✃   Btm Blade Scissors
   // ☓   Saltire              ♏    Scorpius             ✄   White Scissors
   //                       ♐ Sagittarius               
   // ☚    Black Left point Index        ♑   Capricorn              ✆    Telephone Location Sign
   // ☛    Black Right point Index         ♒   Aquarius                ✇  Tape Drive
   // ☜    White Left point Index        ♓    Pisces                 ✈  Airplane
   // ☝  White Up point Index          ♔  White Chess King          ✉  Envelope
   // ☞    White Right point Index         ♕  White Chess Queen           ✍ Writing H&
   // ☟  White Down point Index       ♖  White Chess Rook         ✎   Btm Right Pencil
   // ☠ Skull & Crossbones         ♗  White Chess Bishop           ✏   Pencil
   // ☡  Caution Sign            ♘  White Chess Knight         ✐   Top Right Pencil
   // ☢    Radioactive Sign           ♙  White Chess Pawn           ✓  Check Mark
   // ✔    Heavy Check Mark           ✬    Black Centre White Star        ❂  Circled Open Centre Eight point Star
   // ✕  Multiplication X          ✭    Outlined Black Star         ❃  Heavy Teardrop Pinwheel Asterisk
   // ✖  Heavy Multiplication X       ✮    Heavy Outlined Black Star      ❄  Snowflake
   // ✗  Ballot X               ✯    Pinwheel Star             ❅  Tight Trifoliate Snowflake
   // ✘  Heavy Ballot X            ✰    Shadowed White Star        ❆  Heavy Chevron Snowflake
   // ✚  Heavy Greek Cross          ✱  Heavy Asterisk           ❇  Sparkle
   // ✛  Open Centre Cross          ✲  Open Centre Asterisk        ❈  Heavy Sparkle
   // ✜  Heavy Open Centre Cross       ✳  Eight Spoked Asterisk          ❉  Balloon Asterisk
   // ✝   Latin Cross               ✴  Eight point Black Star        ❊  Eight Teardrop Asterisk
   // ✞  Shadowed White Latin Cross       ✵  Eight point Pinwheel Star       ❋  Heavy Eight Teardrop Asterisk
   // ✟   Outlined Latin Cross          ✶  Six point Black Star         ❍    Shadowed White Circle
   // ✠  Maltese Cross            ✷  Eight point Rectilinear Black Star   ❏  Btm Right Shadowed White Square
   // ✡  Star Of David           ✸  Heavy Eight point Black Star     ❐  Top Right Shadowed White Square
   // ✢  Four Teardrop Asterisk         ✹  Twelve point Black Star        ❑  Btm Right Shadowed White Square
   // ✣  Four Balloon Asterisk         ✺  Sixteen point Asterisk        ❒  Top Right Shadowed White Square
   // ✤  Heavy Four Balloon Asterisk      ✻  Teardrop Asterisk            ❖  Black Diamond Minus White X
   // ✥  Four Club Asterisk           ✼  Open Centre Teardrop Asterisk      
   // ✦  Black Four point Star         ✽  Heavy Teardrop Asterisk         ❛   Heavy Single Turned Comma quote 
   // ✧  White Four point Star         ✾  Six Petalled Black & White Florette    ❜   Heavy Single Comma quote 
   // ✩    Stress Outlined White Star        ✿  Black Florette             ❝  Heavy dbl Turned Comma quote 
   // ✪  Circled White Star            ❀  White Florette             ❞  Heavy dbl Comma quote 
   // ✫    Open Centre Black Star        ❁  Eight Petalled Black Florette     
   // 
   // 
   // ██████████████ █ █ █ █  END   █ █ █ █ ██████████████
END_REGION

REGION Network 18: Special characters — Common character widths and additional whitespace characters
   // ▀▀▀▀▀▀▀▀▀▀▀▀▀▀▀▀▀▀▀▀▀▀▀▀▀▀▀▀▀▀▀▀▀▀▀▀▀▀▀▀▀▀▀▀
   // 
   // TITLE:    COMMON CHARACTER WIDTHS AND ADDITIONAL WHITESPACE CHARACTERS
   // 
   // ▄▄▄▄▄▄▄▄▄▄▄▄▄▄▄▄▄▄▄▄▄▄▄▄▄▄▄▄▄▄▄▄▄▄▄▄▄▄▄▄▄▄▄▄
   // 
   // 
   // This section contains a list of the alphanumeric characters and common punctuation in terms of
   // character width (thinnest first).
   // 
   // The average character widths for each group are based on the frequency of letter usage in 
   // standard (British) English.
   // 
   // The additional whitespace characters complete the set of TIA Portal whitespace characters, these
   // are included for completeness, but duplicate the widths of the standard whitespace characters 
   // listed in previous sections.
   // 
   // 
   // 
   // ▄▄▄▄▄▄▄▄▄▄▄▄▄▄▄▄▄▄▄▄▄▄▄▄▄▄▄▄▄▄▄▄▄▄▄▄▄▄▄▄▄▄▄▄
   // NORMAL CHARACTERS BY WIDTH
   // 
   // 
   // ▐I▌1sp
   // ▐J▌1⅓ sp
   // ▐T▌1⅔ SP
   // ▐F▌2 sp
   // ▐L▌2 sp
   // ▐P▌2 sp
   // ▐R▌2 sp
   // ▐A▌2⅓ SP
   // ▐B▌2⅓ SP
   // ▐C▌2⅓ SP
   // ▐E▌2⅓3 SP
   // ▐K▌2⅓ SP
   // ▐S▌2⅓ SP
   // ▐V▌2⅓ SP
   // ▐X▌2⅓ SP
   // ▐Y▌2⅓ SP
   // ▐Z▌2⅓ SP
   // ▐D▌2⅔ sp
   // ▐G▌2⅔ sp
   // ▐H▌2⅔ sp
   // ▐N▌2⅔ sp
   // ▐U▌2⅔ sp
   // ▐M▌3 sp
   // ▐O▌3 sp
   // ▐Q▌3 sp
   // ▐W▌3 sp
   // Upper avg. (based on frequency and width) = 2.25 normal spaces
   // 
   // ▐f▌1 sp
   // ▐i▌1 sp
   // ▐j▌1 sp
   // ▐l▌1 sp
   // ▐r▌1⅓ sp
   // ▐t▌1⅓ sp
   // ▐x▌1⅔ sp
   // ▐y▌1⅔ sp
   // ▐z▌1⅔ sp
   // ▐c▌2 sp
   // ▐k▌2 sp
   // ▐s▌2 sp
   // ▐v▌2 sp
   // ▐a▌2⅓ sp
   // ▐b▌2⅓ sp
   // ▐d▌2⅓ sp
   // ▐e▌2⅓ sp
   // ▐g▌2⅓ sp
   // ▐h▌2⅓ sp
   // ▐n▌2⅓ sp
   // ▐o▌2⅓ sp
   // ▐p▌2⅓ sp
   // ▐q▌2⅓ sp
   // ▐u▌2⅓ sp
   // ▐w▌3 sp
   // ▐m▌3⅔ sp
   // Lower avg. (based on frequency and width) = 2.00 normal spaces
   // 
   // ▐0▌2⅓ sp
   // ▐1▌2⅓ sp
   // ▐2▌2⅓ sp
   // ▐3▌2⅓ sp
   // ▐4▌2⅓ sp
   // ▐5▌2⅓ sp
   // ▐6▌2⅓ sp
   // ▐7▌2⅓ sp
   // ▐8▌2⅓ sp
   // ▐9▌2⅓ sp
   // Numbers = 2.33 sp
   // 
   // ▐!▌1 sp
   // ▐'▌1 sp
   // ▐,▌1 sp
   // ▐-▌1 sp
   // ▐.▌1 sp
   // ▐/▌1 sp
   // ▐\▌1 sp
   // ▐|▌1 sp
   // ▐[▌1⅓ sp
   // ▐]▌1⅓ sp
   // ▐:▌1⅓ sp
   // ▐:▌1⅓ sp
   // ▐(▌1⅓ sp
   // ▐)▌1⅓ sp
   // ▐{▌1⅔ sp
   // ▐}▌1⅔ sp
   // ▐"▌1⅔ sp
   // ▐?▌1⅔ sp
   // ▐<▌2 sp
   // ▐>▌2 sp
   // ▐^▌2 sp
   // ▐_▌2 sp
   // ▐~▌2 sp
   // ▐=▌2⅓ sp
   // ▐$▌2⅓ sp
   // ▐*▌2⅓ sp
   // ▐+▌2⅓ sp
   // ▐`▌2⅓ sp
   // ▐&▌2⅔ sp
   // ▐#▌2⅔ sp
   // ▐%▌3 sp
   // ▐@▌3⅓ sp
   // Punctuation avg. 1 sp (based on comma, full stop and dash being the most common)
   // 
   // 
   // 
   // ▄▄▄▄▄▄▄▄▄▄▄▄▄▄▄▄▄▄▄▄▄▄▄▄▄▄▄▄▄▄▄▄▄▄▄▄▄▄▄▄▄▄▄▄
   // ALL OTHER WHITESPACE CHARACTERS
   // 
   // The other whitespace characters (Hair space, figure space &c.) are supported by the Siemens
   // font, but have the identical widths to those listed above. The full list is shown below:
   // 
   // ▐  ▌2 Em spaces
   // ▐    ▌4 En space      (1/2 em)
   // ▐      ▌6 Three per em     (1/3 em)
   // ▐        ▌8 Punctuation space (1/4 em)
   // ▐        ▌8 Normal space      (1/4 em)
   // ▐        ▌8 Four per em      (1/4 em)
   // ▐        ▌8 Figure space     (1/4 em)
   // ▐            ▌12 Six per em    (1/6 em)
   // ▐            ▌12 Hair space       (1/6 em)
   // 
   //                 ━━━  ⬙⬙⬙⬙⬙⬙  ━━━
   // 
   // 
   // ██████████████ █ █ █ █  END   █ █ █ █ ██████████████
END_REGION

REGION Network 19: OB1 NETWORK 1 — Project description
   // ▀▀▀▀▀▀▀▀▀▀▀▀▀▀▀▀▀▀▀▀▀▀▀▀▀▀▀▀▀▀▀▀▀▀▀▀▀▀▀▀▀▀▀▀
   // 
   // TITLE:    PS2001 — PRACTICAL SERIES AUTOMATION LIBRARY
   // 
   // ▄▄▄▄▄▄▄▄▄▄▄▄▄▄▄▄▄▄▄▄▄▄▄▄▄▄▄▄▄▄▄▄▄▄▄▄▄▄▄▄▄▄▄▄
   // 
   // 
   // ――――――――――――――――――――――――――――――――――
   // COPYRIGHT:       © 2020 Michael Gledhill
   //           Part of the Practical Series of Publications
   //           Published in the United Kingdom
   //           mg@practicalseries.com
   //           https://practicalseries.com
   // ――――――――――――――――――――――――――――――――――
   // CUSTOMER:       Practical Series of Publications (PSP)
   // 
   // PROJECT:      Practical Series Automation Library (PAL)
   // 
   // PROJECT NO.:       PS2001
   // ――――――――――――――――――――――――――――――――――
   // CONTROLLER:       CPU 1515-2PN/DP
   // 
   // CONTROLLER NAME:    CON100
   // 
   // IP ADDRESS:      192.168.001.100
   // ――――――――――――――――――――――――――――――――――
   // TIA PROJECT NAME:    PS2001-PAL-D0000
   // 
   // STATUS:        DEVELOPMENT
   // ――――――――――――――――――――――――――――――――――
   // PROTECTION:     To minimise the risk of inadvertent modification to 
   //           tested modules, certain blocks will be released for 
   //           use with “protected access” (referred to a “write 
   //           protection” in Siemens terminology), this allows the 
   //           block to be used normally, but prevents the block 
   //           being accidentally modified. 
   // 
   //           This is in accordance with the risk assessment given 
   //           in the Validation Plant (VP), Appendix A [Ref. 002].
   // 
   //           ┌─────────────────────┐
   //           │ THE WRITE PROTECTION PASSWORD IS: PS2001 │
   //           └─────────────────────┘
   // 
   // 
   // ▄▄▄▄▄▄▄▄▄▄▄▄▄▄▄▄▄▄▄▄▄▄▄▄▄▄▄▄▄▄▄▄▄▄▄▄▄▄▄▄▄▄▄▄
   // PROJECT OVERVIEW
   // 
   // 
   // The PAL is a library of software modules and templates that have been developed for the 
   // Siemens Simatic S7-1500 range of controllers (and to a lesser extent the S7-1200 range).
   // 
   // The full library and all necessary documentation is available from the Practical Series website:
   // 
   //      https://practicalseries.com/2001-pal/index.html
   // 
   // 
   // The PAL is configured and deployed using the Siemens Simatic TIA Portal programming 
   // environment.
   // 
   // The PAL software structure is designed such that it is applicable to virtually all industrial 
   // applications that can generally controlled by a programmable logic controller.
   // 
   // The PAL software being developed as part of this Project, is considered to be suitable for use in 
   // the following types of industries (this is not an exhaustive list):
   // 
   //    •   Water and waste water treatment
   //    •   Pharmaceutical and batch production
   //    •   Brewing and fermentation
   //    •   Chemical manufacturing
   //    •   Oil and gas systems
   //    •   Food and beverage production
   // 
   // Such applications can generally be thought of as processes that operate with a response time
   // of more than 100 ms. I.e. the system would not be expected to respond to some stimuli faster
   // than 100 ms. In practice, a Controller may (and usually will) respond faster than this; however, 
   // a response time of 100 ms is considered to be an acceptable limit for PLC control.
   // 
   // At its most basic level, the PAL will be a library of software modules that control the fundamental 
   // aspects of an industrial plant; such modules would for example read the value of an instrument, 
   // operate a valve or drive, perform a calculation &c.
   // 
   // Such software modules are referred to as standard modules, these are fixed modules that 
   // perform a particular function and are identical across all software installations.
   // 
   // The PAL also contains application specific modules; these contain software that is applicable 
   // to the plant being controlled.
   // 
   // The Practical Series Automation Library is freely available under the MIT Open Source licence 
   // (see below). Those who find it useful may, if they wish, make a donation to support the library. 
   // 
   // Donations can be made here:
   // 
   //      https://practicalseries.com/2001-pal/11-web/81-00-pay.html
   // 
   // The PAL contains fully deployable software that has been developed by the author in his 
   // profession as a chartered electrical engineer. It is currently in use on various live plants 
   // throughout the UK and in some other parts of the world. 
   // 
   // This software is suitable for controlling and automating most industrial applications (typical 
   // process applications). It is easy to use and configure, but does have a degree of practical 
   // complexity appropriate for the environments within which it is employed. It is heavily 
   // configurable, has various operating modes and is suitable for a multitude of industrial 
   // applications.
   // 
   // IF YOU DON’T UNDERSTAND IT, DON’T USE IT. IF YOU DO USE IT, YOU DO SO AT YOUR OWN RISK.
   // 
   //                ━━━   ⬙⬙⬙⬙⬙⬙   ━━━
   // 
   // ▄▄▄▄▄▄▄▄▄▄▄▄▄▄▄▄▄▄▄▄▄▄▄▄▄▄▄▄▄▄▄▄▄▄▄▄▄▄▄▄▄▄▄▄
   // DOCUMENT REFERENCES
   // 
   //  ――――――――――――――――――――――――――――――――――――――――――
   //  REF.     DOCUMENT NO.       TITLE
   //  ――――――――――――――――――――――――――――――――――――――――――
   //  001  PS2001-5-0101-001   Quality Plan (QP)
   //  002  PS2001-5-0121-002   Validation Plan (VP)
   //  003  PS2001-5-0131-003   Test Plan (TP)
   //  004  PS2001-5-1101-001   User requirements specification (URS)
   //  005  PS2001-5-1111-001   Requirement Traceability Matrix (RTM)
   //  006  PS2001-5-2101-001   Functional Specification (FS) 
   //  007  PS2001-5-2211-001   Hardware Design Specification (HDS)
   //  008  PS2001-5-2311-001   Software Design Specification (SDS)
   //  009  PS2001-5-7111-001   User Guide (UG)
   //  010  PS2001-5-2313-011   Style Guide (SG)
   //  011  PS2001-5-2312-fcNo.    Software Module Design Specification (SMDS)
   //  012  PS2001-5-2301-001   Software Module Register (SMR)
   //  013  PS2001-5-2302-011   Software Control and Mechanism (SCM)
   //  ――――――――――――――――――――――――――――――――――――――――――
   // 
   //                ━━━   ⬙⬙⬙⬙⬙⬙   ━━━
   // 
   // 
   // ▄▄▄▄▄▄▄▄▄▄▄▄▄▄▄▄▄▄▄▄▄▄▄▄▄▄▄▄▄▄▄▄▄▄▄▄▄▄▄▄▄▄▄▄
   // COMPLETED MODULES 
   // 
   // COMPLETED MODULES 
   // 
   //  ――――――――――――――――――――-―-- STATIC DATA       ― DYNAMIC  DAT A   ―
   //  BLOCK     NAME         REVISION    UDT/DB    REVISION  UDT/DB    REVISION  
   //  ――――――――――――――――――――――――――――――――――――――――――
   //  FC01001 StdSysGlobalData      001.000   UT 01000   001.000-R UT 21000   001.000-R
   //                  2020-11-20   UT 01001   001.000-R UT 21000   001.000-R 
   //                           None           DB21000   001.000-R
   //  ――――――――――――――――――――――――――――――――――――――――――
   //  FC02001 StdInstAnalogRead    001.000   UT 02001   001.000-R UT 22001   001.000-R
   //                  2020-11-20   DB02001   001.000-R DB22001   001.000-R
   //  ――――――――――――――――――――――――――――――――――――――――――
   //  FC18001 StdSubScaleAI      001.000   None           None 
   //                  2020-12-09   None           None
   //  ――――――――――――――――――――――――――――――――――――――――――
   //  FC18151 StdSubTimeEventRTC   001.000   None           UT 38151   001.000-R
   //                  2020-11-20                  DB38151   001.000-R
   //  ――――――――――――――――――――――――――――――――――――――――――
   //  FC61000 DocGenExample     001.000   None           None 
   //                  2020-11-20   None           None          
   //  ――――――――――――――――――――――――――――――――――――――――――
   //  FC21000 AppSys          001.000   None           None 
   //                  2020-12-04   None           None          
   //  ――――――――――――――――――――――――――――――――――――――――――
   //  See Software Module Register [Ref. 012] for full details
   // 
   //                ━━━   ⬙⬙⬙⬙⬙⬙   ━━━
   // 
   // 
   // ▀▀▀▀▀▀▀▀▀▀▀▀▀▀▀▀▀▀▀▀▀▀▀▀▀▀▀▀▀▀▀▀▀▀▀▀▀▀▀▀▀▀▀▀
   // LICENCE AND CONTACT INFORMATION
   // 
   // This software and its associated documentation is made available under the MIT Licence:
   // 
   // ════════════════════════════════════════════
   // 
   // The MIT License (MIT)
   // 
   // Copyright © 2020 Michael Gledhill
   // 
   // Permission is hereby granted, free of charge, to any person obtaining a copy of this software 
   // and associated documentation files (the “Software”), to deal in the Software without restriction, 
   // including without limitation the rights to use, copy, modify, merge, publish, distribute, 
   // sublicense, and/or sell copies of the Software, and to permit persons to whom the Software is 
   // furnished to do so, subject to the following conditions: 
   // 
   // The above copyright notice and this permission notice shall be included in all copies or 
   // substantial portions of the Software.
   // 
   // THE SOFTWARE IS PROVIDED “AS IS”, WITHOUT WARRANTY OF ANY KIND, EXPRESS OR IMPLIED, 
   // INCLUDING BUT NOT LIMITED TO THE WARRANTIES OF MERCHANTABILITY, FITNESS FOR A 
   // PARTICULAR PURPOSE AND NON-INFRINGEMENT. IN NO EVENT SHALL THE AUTHORS OR COPYRIGHT 
   // HOLDERS BE LIABLE FOR ANY CLAIM, DAMAGES OR OTHER LIABILITY, WHETHER IN AN ACTION OF 
   // CONTRACT, TORT OR OTHERWISE, ARISING FROM, OUT OF OR IN CONNECTION WITH THE SOFTWARE 
   // OR THE USE OR OTHER DEALINGS IN THE SOFTWARE.
   // 
   // ════════════════════════════════════════════
   //                    ┌────────────┐
   // You can reach the author by email here:   │  mg@practicalseries.com  │
   //                    └────────────┘
   // Questions, corrections, constructive criticism and complaints (polite ones) are invited.
   // 
   // ▄▄▄▄▄▄▄▄▄▄▄▄▄▄▄▄▄▄▄▄▄▄▄▄▄▄▄▄▄▄▄▄▄▄▄▄▄▄▄▄▄▄▄▄
   // 
   // 
   //                ━━━   ⬙⬙⬙⬙⬙⬙   ━━━
   // 
   // 
   // 
   // ██████████████ █ █ █ █  END   █ █ █ █ ██████████████
END_REGION

REGION Network 20: OB1 NETWORK 2 — Current revision and modification history
   // ▄▄▄▄▄▄▄▄▄▄▄▄▄▄▄▄▄▄▄▄▄▄▄▄▄▄▄▄▄▄▄▄▄▄▄▄▄▄▄▄▄▄▄▄
   // MODIFICATION HISTORY (GITHUB VERSION CONTROL SYSTEM)
   // 
   // 
   // This is a complete summary of all primary software modifications (commit points) made to this 
   // TIA Portal project (the latest commit tag is at the top of the list). 
   // 
   // The latest commit tag, author and the date of the revision are hardcoded into the Controller in 
   // this network (allowing revision data to be obtained directly from the Controller).
   // 
   // The development of the software project is stored and managed within the GIT Source Code 
   // Management system (a version control system or VCS) in conjunction with the GitHub online 
   // hosting system. The software in its entirety is available in the GitHub remote repository:
   // 
   //      https://github.com/practicalseries/PS2001-pal-software
   // 
   // This repository is public and can be freely “forked” (copied) and used under the MIT Licence.
   // The MIT Licence is reproduced in full in the previous network.
   // 
   //  ———————————————————————————————————————————
   //  DATE     COMMIT TAG       AUTHOR        REASON FOR MODIFICATION
   //  ———————————————————————————————————————————
   //  2021.02.02    D0002      M. Gledhill      Baseline build
   // 
   //  2021.02.02    D0001      M. Gledhill      Hardware build
   // 
   //  2021.02.02    D0000      M. Gledhill      Initial commit — repository created
   //  ———————————————————————————————————————————
   // 
   // 
   // ▄▄▄▄▄▄▄▄▄▄▄▄▄▄▄▄▄▄▄▄▄▄▄▄▄▄▄▄▄▄▄▄▄▄▄▄▄▄▄▄▄▄▄▄
   RUNG wire#powerrail
      I_Contact( #_FALSE )
      wire#w1
      S_Move(in := 'PS2001', out => #revInfo.REV_BLOCK)
   END_RUNG
   RUNG wire#w1
      S_Move(in := '001.000-R', out => #revInfo.REV_NUMBER)
   END_RUNG
   RUNG wire#w1
      S_Move(in := '2020.10.20', out => #revInfo.REV_DATE)
   END_RUNG
   RUNG wire#w1
      S_Move(in := 'M. Gledhill', out => #revInfo.REV_AUTHOR)
   END_RUNG
   // the same network as SCL:
   IF NOT #_FALSE THEN
       #revInfo.REV_BLOCK := 'PS2001';
       #revInfo.REV_NUMBER := '001.000-R';
       #revInfo.REV_DATE := '2020.10.20';
       #revInfo.REV_AUTHOR := 'M. Gledhill';
   END_IF;
END_REGION

REGION Network 21: Load the system RTC and store in local variable [typical network comment]
   // ▀▀▀▀▀▀▀▀▀▀▀▀▀▀▀▀▀▀▀▀▀▀▀▀▀▀▀▀▀▀▀▀▀▀▀▀▀▀▀▀▀▀▀▀
   // The system block RD_SYS_T reads the time of day, the date and the day of week from the system 
   // real time clock as a DTL (or Date_And_Time_Long) data type (one just being the shorthand 
   // notation of the other). The result is stored in a local variable for decoding.
   // 
   // The DTL data type stores the date and time information in 8 consecutive bytes in BCD format 
   // as follows:
   // 
   // 
   //  ――――――――――――――――――――――――――――――――――――――――――
   //  DATA         DESCRIPTION
   // 
   //  0          Dear        (00h-89h = 2000 to 2089)   (90h-99h = 1990 to 1999)
   //  1          Month      (00h-12h = Jan to Dec)
   //  2          Day       (01h-31h)
   //  3          Hour        (00h-23h)
   //  4          Minute        (00h-59h)
   //  5          Month      (00h-12h = Jan to Dec)
   //  6-7         Millisecond      Uses byte 6 and most significant 4 bits of byte 7)
   //  7          Day of Week    least significant 4 bits (1h-7h = Sun to Sat)
   //  ――――――――――――――――――――――――――――――――――――――――――
   // 
   // 
   // The local variable is of type DTL (Date_And_Time_Long), this is compatible with the DT output
   // from RD_SYST, but allows the individual elements of the DT structure to be accesses
   // individually as symbols.
   // 
   // Note:    The DTL format can store more information (it can for example handle years in the 
   //      range 1970 to 2262; however, it will still only store the data in the table above
   //      when used with RS_SYS_T. 
   // ▄▄▄▄▄▄▄▄▄▄▄▄▄▄▄▄▄▄▄▄▄▄▄▄▄▄▄▄▄▄▄▄▄▄▄▄▄▄▄▄▄▄▄▄
END_REGION

REGION Network 22: ██ STEP 03340 — DECLARATION (RUNNING) [sequence network comment]
   // ▀▀▀▀▀▀▀▀▀▀▀▀▀▀▀▀▀▀▀▀▀▀▀▀▀▀▀▀▀▀▀▀▀▀▀▀▀▀▀▀▀▀▀▀
   // 
   //  ███   ███   ███  █  █   ███  
   // █   █ █   █ █   █ █  █  █   █ 
   // █  ██     █     █ █  █  █  ██ 
   // █ █ █  ███   ███  █████ █ █ █ 
   // ██  █     █     █    █  ██  █ 
   // █   █ █   █ █   █    █  █   █ 
   //  ███   ███   ███     █   ███  
   // 
   // ▄▄▄▄▄▄▄▄▄▄▄▄▄▄▄▄▄▄▄▄▄▄▄▄▄▄▄▄▄▄▄▄▄▄▄▄▄▄▄▄▄▄▄▄
   // STEP DESCRIPTION
   // 
   // 
   // Open the dry air purge valve (SV4201), activate the operator prompt ABORT PURGE.
   // 
   // If the main chamber humidity level falls below the target value proceed to the next step.
   // 
   // If the operator presses the ABORT PURGE button proceed to step 03400.
   // 
   // 
   // 
   // ▄▄▄▄▄▄▄▄▄▄▄▄▄▄▄▄▄▄▄▄▄▄▄▄▄▄▄▄▄▄▄▄▄▄▄▄▄▄▄▄▄▄▄▄
   // STEP PHASE AND DELAY CONDITIONS
   // 
   // 
   //  ――――――――――――――――――――――――――――――――――――――――――
   //  PHASE         ACTION
   //  ――――――――――――――――――――――――――――――――――――――――――
   //  INITIALISING      Activate the ABORT PURGE enable signal
   // 
   //  PROCESSING    Open SV4201
   // 
   //  TERMINATING    Clear the ABORT PURGE enable signal and any ABORT PURGE pressed
   //           signal
   // 
   //  STEP DELAY      No delay
   //  ――――――――――――――――――――――――――――――――――――――――――
   // 
   // 
   // 
   // ▄▄▄▄▄▄▄▄▄▄▄▄▄▄▄▄▄▄▄▄▄▄▄▄▄▄▄▄▄▄▄▄▄▄▄▄▄▄▄▄▄▄▄▄
   // STEP TRANSITION CONDITIONS
   // 
   // 
   //  ――――――――――――――――――――――――――――――――――――――――――
   //  TRANSITION      TO STEP    TRANSITION CONDITIONS
   //  ――――――――――――――――――――――――――――――――――――――――――
   //  1.        03350      HIC001 ≤ HUMIDITY_LIMIT
   // 
   //  2.        03400      Operator has pressed ABORT PURGE button
   //  ――――――――――――――――――――――――――――――――――――――――――
   // 
   // 
   // ▄▄▄▄▄▄▄▄▄▄▄▄▄▄▄▄▄▄▄▄▄▄▄▄▄▄▄▄▄▄▄▄▄▄▄▄▄▄▄▄▄▄▄▄
END_REGION

REGION Network 23: STEP 03340 — ACTION (INITIALISE) [sequence network comment]
   // ▀▀▀▀▀▀▀▀▀▀▀▀▀▀▀▀▀▀▀▀▀▀▀▀▀▀▀▀▀▀▀▀▀▀▀▀▀▀▀▀▀▀▀▀
   // INITIALISE PHASE
   // 
   // Activate the ABORT PURGE enable signal
   // (this is a temporary signal passed to the handling DB at the end of the block)
   // ▄▄▄▄▄▄▄▄▄▄▄▄▄▄▄▄▄▄▄▄▄▄▄▄▄▄▄▄▄▄▄▄▄▄▄▄▄▄▄▄▄▄▄▄
END_REGION

REGION Network 24: STEP 03340 — TRANSITION 01 [sequence network comment]
   // ▀▀▀▀▀▀▀▀▀▀▀▀▀▀▀▀▀▀▀▀▀▀▀▀▀▀▀▀▀▀▀▀▀▀▀▀▀▀▀▀▀▀▀▀
   // TRANSITION CONDITION 01
   // 
   // Wait for humidity to reach target level HIC001 ≤ HUMIDITY_LIMIT
   // ▄▄▄▄▄▄▄▄▄▄▄▄▄▄▄▄▄▄▄▄▄▄▄▄▄▄▄▄▄▄▄▄▄▄▄▄▄▄▄▄▄▄▄▄
END_REGION

REGION Network 25: LICENCE AND CONTACT INFORMATION [final network]
   // ▀▀▀▀▀▀▀▀▀▀▀▀▀▀▀▀▀▀▀▀▀▀▀▀▀▀▀▀▀▀▀▀▀▀▀▀▀▀▀▀▀▀▀▀
   // LICENCE AND CONTACT INFORMATION
   // 
   // This software and its associated documentation is made available under the MIT Licence:
   // 
   // ════════════════════════════════════════════
   // 
   // The MIT License (MIT)
   // 
   // Copyright © 2020 Michael Gledhill
   // 
   // Permission is hereby granted, free of charge, to any person obtaining a copy of this software 
   // and associated documentation files (the “Software”), to deal in the Software without restriction, 
   // including without limitation the rights to use, copy, modify, merge, publish, distribute, 
   // sublicense, and/or sell copies of the Software, and to permit persons to whom the Software is 
   // furnished to do so, subject to the following conditions: 
   // 
   // The above copyright notice and this permission notice shall be included in all copies or 
   // substantial portions of the Software.
   // 
   // THE SOFTWARE IS PROVIDED “AS IS”, WITHOUT WARRANTY OF ANY KIND, EXPRESS OR IMPLIED, 
   // INCLUDING BUT NOT LIMITED TO THE WARRANTIES OF MERCHANTABILITY, FITNESS FOR A 
   // PARTICULAR PURPOSE AND NON-INFRINGEMENT. IN NO EVENT SHALL THE AUTHORS OR COPYRIGHT 
   // HOLDERS BE LIABLE FOR ANY CLAIM, DAMAGES OR OTHER LIABILITY, WHETHER IN AN ACTION OF 
   // CONTRACT, TORT OR OTHERWISE, ARISING FROM, OUT OF OR IN CONNECTION WITH THE SOFTWARE 
   // OR THE USE OR OTHER DEALINGS IN THE SOFTWARE.
   // 
   // ════════════════════════════════════════════
   //                    ┌────────────┐
   // You can reach the author by email here:   │  mg@practicalseries.com  │
   //                    └────────────┘
   // Questions, corrections, constructive criticism and complaints (polite ones) are invited.
   // 
   // ▄▄▄▄▄▄▄▄▄▄▄▄▄▄▄▄▄▄▄▄▄▄▄▄▄▄▄▄▄▄▄▄▄▄▄▄▄▄▄▄▄▄▄▄
   RUNG wire#powerrail
      I_Contact( #_FALSE )
      wire#w1
      S_Move(in := 'MIT LICENSE', out => #licInfo.LICENCE_TYPE)
   END_RUNG
   RUNG wire#w1
      S_Move(in := '2020 Michael Gledhill', out => #licInfo.COPYRIGHT)
   END_RUNG
   // the same network as SCL:
   IF NOT #_FALSE THEN
       #licInfo.LICENCE_TYPE := 'MIT LICENSE';
       #licInfo.COPYRIGHT := '2020 Michael Gledhill';
   END_IF;
END_REGION
END_FUNCTION

FUNCTION "FC01001_StdSysGlobalData" : Void   // FC1001, LAD
TITLE = Standard - Sys — Global Data
{ S7_Optimized_Access := 'TRUE' }
AUTHOR : M_Gledhill
FAMILY : System
NAME : StdSysGlobalData
VERSION : 1.0
// PRACTICAL SERIES AUTOMATION LIBRARY (PAL)   —   COPYRIGHT 2020 – M. GLEDHILL (MIT LICENCE)
//                   ———— ◆ ————
//  FOR DETAILED DOCUMENTATION — SELECT THE BLOCK IN THE PROJECT TREE AND PRESS SHIFT + F1
//  FULL ONLINE DOCUMENTATION IS AVAILABLE AT: https://practicalseries.com/2001-pal/index.html
// stored: AutoNumber false, IsIECCheckEnabled false, SetENOAutomatically false, UDAEnableTagReadback false
   VAR_INPUT
      CLOCK_MEM : Byte;   // The clock memory byte (within the PAL this is always MB10)
   END_VAR
   VAR_OUTPUT
      SYS_SIGNAL_TAGS : Int;   // The system logic and timing signals for direct access
   END_VAR
   VAR_IN_OUT
      SYS_SIGNALS : "UT21000_Dy_SysSignals";   // The system logic and timing signals for parametric access
      SYS_DATA : "UT21001_Dy_SysData";   // The system data storage structure interface, holds the cycle & RTC data
   END_VAR
   VAR_TEMP
      revInfo : "UT01000_St_SysRevision";   // Revision information for this block
      licInfo : "UT01001_St_SysLicence";   // Licence information for this block
      SI_ProgramCycle : SI_ProgramCycle;   // Used by RD_SINFO, holds information for the current OB
      SI_StartUp : SI_Startup;   // Used by RD_SINFO, holds information for the last start-up OB
      wrkInt : Int;   // Working storage (integer)
      wrkDInt : DInt;   // Working storage (double integer)
      wrkReal : Real;   // Working storage (real)
      wrkLTime : LTime;   // Working storage (Long Time)
      wrkDTL : DTL;   // Working storage (DateTimeLong)
   END_VAR
   VAR_TEMP   // added for the SCL form of the ladder/FBD networks
      _w1 : Bool;
      _w2 : Bool;
      _w3 : Bool;
      _w4 : Bool;
      _w5 : Bool;
      _w6 : Bool;
   END_VAR
BEGIN

